FUNCTION_BLOCK Hutschienenmoped_XL_8_PWM (* Service Interface Function Block Type *)
  (* Function: All Outputs; Description: this maps to QD this is a PWM Out. Will immediately go to the Desired Duty Cycle. *)
  (* Version 1.0, 2018-12-05, Jose Cabral *)
  (* Version 1.1, 2022-08-04, Franz Höpfinger, HR Agrartechnik GmbH *)
  (* Version 1.2, 2023-01-05, Franz Höpfinger, HR Agrartechnik GmbH *)
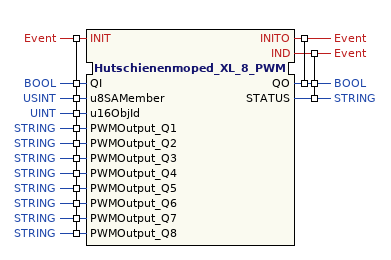
  EVENT_INPUT
    INIT WITH QI, u8SAMember, u16ObjId, PWMOutput_Q1, PWMOutput_Q2, PWMOutput_Q3, PWMOutput_Q4, PWMOutput_Q5, PWMOutput_Q6, PWMOutput_Q7, PWMOutput_Q8; (* Service Initialization *)
  END_EVENT
  EVENT_OUTPUT
    INITO WITH QO; (* Initialization Confirm *)
    IND WITH QO, STATUS; (* Indication from Resource *)
  END_EVENT
  VAR_INPUT
    QI : BOOL; (* Event Input Qualifier *)
    u8SAMember : USINT := GLOBAL; (* Dummy !, set to GLOBAL if in doubt. OFF deactivates FB. *)
    u16ObjId : UINT := ID_NULL; (* Dummy ! set to ID_NULL if in Doubt. ID_OFF deactivates FB. *)
    PWMOutput_Q1 : STRING;
    PWMOutput_Q2 : STRING;
    PWMOutput_Q3 : STRING;
    PWMOutput_Q4 : STRING;
    PWMOutput_Q5 : STRING;
    PWMOutput_Q6 : STRING;
    PWMOutput_Q7 : STRING;
    PWMOutput_Q8 : STRING;
  END_VAR
  VAR_OUTPUT
    QO : BOOL; (* Event Output Qualifier *)
    STATUS : STRING; (* Service Status *)
  END_VAR
END_FUNCTION_BLOCK
